// TIA Portal project "Homework Day8" (V15)

(* hardware
DEVICE "S7-1200 station_1"  S7-1200 Station
   slot 0: "Rack_0"  S7-1200 Rack  Rack  V1.0
   slot 1: "PLC_1"  CPU 1215C AC/DC/Rly  6ES7 215-1BG40-0XB0  V4.0
*)

// ===== PLC "PLC_1"  CPU 1215C AC/DC/Rly =====

VAR_GLOBAL   // PLC tag table "VARIB"
   "Start" AT %M0.0 : Bool;
   "Stop" AT %M0.1 : Bool;
   "Process" AT %M0.2 : Bool;
   "Temp Value" AT %MW64 : Word;
   "Temp Value Norm" AT %MD10 : Real;
   "Temp Actual" AT %MD14 : Real;
   "Error" AT %MD18 : Real;
   "Heater" AT %Q0.0 : Bool;
   "Flash" AT %M0.3 : Bool;
   "Turn On" AT %M0.4 : Bool;
   "Turn Off" AT %M0.5 : Bool;
   "again" AT %M0.6 : Bool;
   "Sample 1" AT %MD100 : Real;
   "Sample 2" AT %MD104 : Real;
   "Sample 3" AT %MD108 : Real;
   "Sample 4" AT %MD112 : Real;
   "Sample 5" AT %MD116 : Real;
   "Sample Pulse" AT %M0.7 : Bool;
   "Edge Bit" AT %M1.0 : Bool;
   "Average Temperature" AT %MD22 : Real;
END_VAR

// folder: System blocks/Program resources

DATA_BLOCK "Timer 3"   // DB1
{ S7_Optimized_Access := 'TRUE' }
AUTHOR : Simatic
FAMILY : IEC
NAME : IEC_TMR
VERSION : 1.0
// stored: InstanceOfName IEC_TIMER
"IEC_TIMER"
BEGIN
END_DATA_BLOCK

DATA_BLOCK "Timer 1"   // DB2
{ S7_Optimized_Access := 'TRUE' }
AUTHOR : Simatic
FAMILY : IEC
NAME : IEC_TMR
VERSION : 1.0
// stored: InstanceOfName IEC_TIMER
"IEC_TIMER"
BEGIN
END_DATA_BLOCK

DATA_BLOCK "Timer 2"   // DB3
{ S7_Optimized_Access := 'TRUE' }
AUTHOR : Simatic
FAMILY : IEC
NAME : IEC_TMR
VERSION : 1.0
// stored: InstanceOfName IEC_TIMER
"IEC_TIMER"
BEGIN
END_DATA_BLOCK

// folder: (top level)

ORGANIZATION_BLOCK "Main"   // OB1, LAD, ProgramCycle
TITLE = "Main Program Sweep (Cycle)"
{ S7_Optimized_Access := 'TRUE' }
VERSION : 0.1
// Temperature Control with PID Simulation (Math, Comparison, Timers)
// 
// Scenario: A heater maintains a temperature setpoint. The current temperature is Temp_Actual (REAL) and the setpoint is Temp_Setpoint (REAL = 75.0°C).
// 
// Requirements:
// 1. Use Math to calculate the error: Error = Temp_Setpoint - Temp_Actual.
// 2. Use Comparison to control the heater:
// • If Error > 5.0, turn heater ON 100% (continuous).
// If Error between 1.0 and 5.0, use a Timer to cycle the heater ON for 5 seconds, OFF for 5 seconds (50% duty cycle).
// • If Error < 1.0, turn heater OFF.
// 3. Use a Timer to sample the temperature every 1 second and store the last 5 samples (use Math to calculate the average)
   VAR_INPUT
      Initial_Call : Bool;   // Initial call of this OB
      Remanence : Bool;   // =True, if remanent data are available
   END_VAR
BEGIN

REGION Network 1
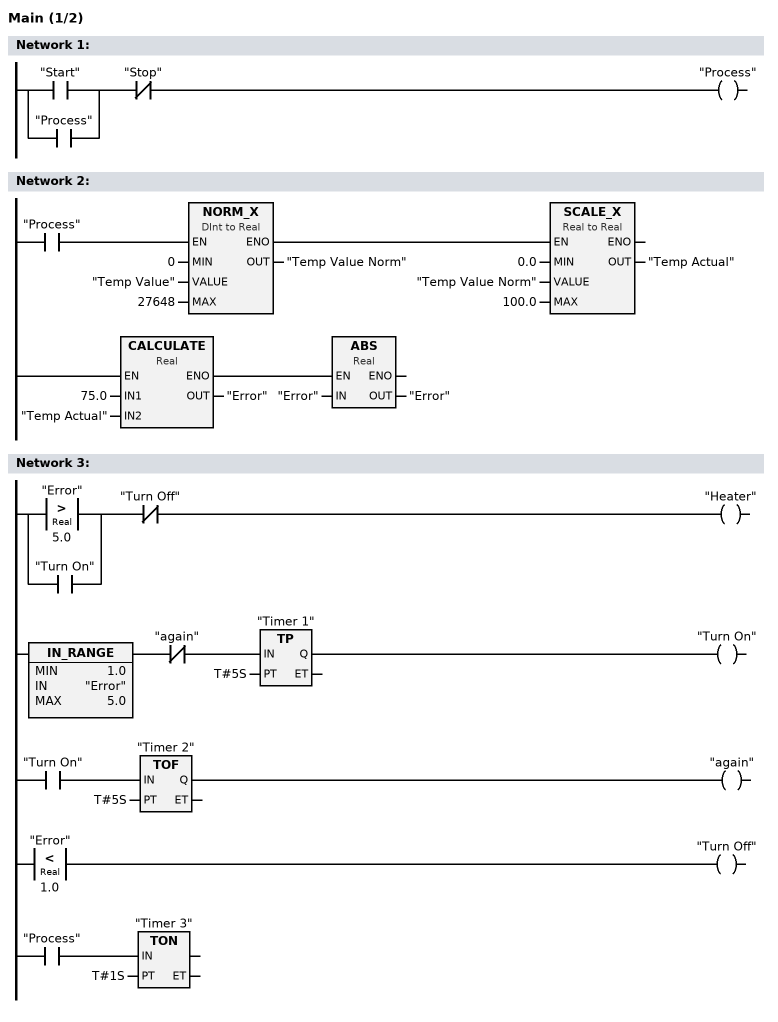
   RUNG wire#powerrail
      Contact( "Start" )
      wire#w1
      I_Contact( "Stop" )
      Coil( "Process" )
   END_RUNG
   RUNG wire#powerrail
      Contact( "Process" )
   END_RUNG wire#w1
   // the same network as SCL:
   "Process" := ("Start" OR "Process") AND NOT "Stop";
END_REGION

REGION Network 2
   RUNG wire#powerrail
      Contact( "Process" )
      { S7_Templates := "[SrcType := DInt, DestType := Real]" } Normalize(min := 0, value := "Temp Value", max := 27648, out => "Temp Value Norm")
      { S7_Templates := "[SrcType := Real, DestType := Real]" } Scale(min := 0.0, value := "Temp Value Norm", max := 100.0, out => "Temp Actual")
   END_RUNG
   RUNG wire#powerrail
      { S7_Templates := "SrcType := Real"; S7_Expression := "IN1-IN2" } Calculate(in1 := 75.0, in2 := "Temp Actual", out => "Error")
      { S7_Templates := "SrcType := Real" } Abs(in := "Error", out => "Error")
   END_RUNG
   // the same network as SCL:
   IF "Process" THEN
       "Temp Value Norm" := NORM_X(MIN := 0, VALUE := "Temp Value", MAX := 27648);
       "Temp Actual" := SCALE_X(MIN := 0.0, VALUE := "Temp Value Norm", MAX := 100.0);
   END_IF;
   "Error" := 75.0-"Temp Actual";
   "Error" := ABS("Error");
END_REGION

REGION Network 3
   "Heater" := (("Error" > 5.0) OR "Turn On") AND NOT "Turn Off";
   "Timer 1".TP(IN := (1.0 <= "Error") AND ("Error" <= 5.0) AND NOT "again", PT := T#5S);
   "Turn On" := "Timer 1".Q;
   "Timer 2".TOF(IN := "Turn On", PT := T#5S);
   "again" := "Timer 2".Q;
   "Turn Off" := "Error" < 1.0;
   "Timer 3".TON(IN := "Process", PT := T#1S);
END_REGION

REGION Network 4
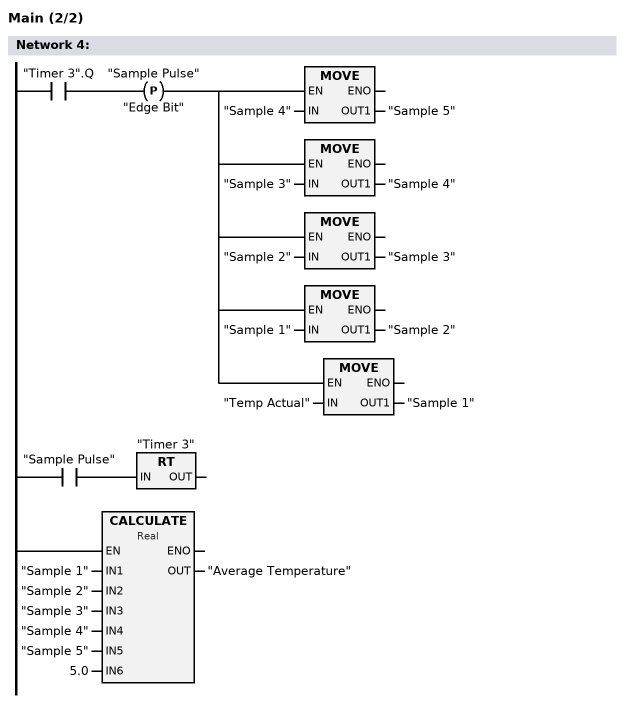
   "Sample Pulse" := "Timer 3".Q AND NOT "Edge Bit";   // rising edge
   "Edge Bit" := "Timer 3".Q;
   IF "Timer 3".Q THEN
       "Sample 5" := "Sample 4";
       "Sample 4" := "Sample 3";
       "Sample 3" := "Sample 2";
       "Sample 2" := "Sample 1";
       "Sample 1" := "Temp Actual";
   END_IF;
   IF "Sample Pulse" THEN RESET_TIMER("Timer 3"); END_IF;
   "Average Temperature" := ("Sample 1"+"Sample 2"+"Sample 3"+"Sample 4"+"Sample 5")/5.0;
END_REGION
END_ORGANIZATION_BLOCK